{attribute 'GeneratedUsingTerminal: EL5122-0000-0016'}
{attribute addProperty BoxType "EL5122-0000-0016"}
{attribute addProperty Description "EL5122 2Ch. Inc. Encoder 5V (2xAB TTL)"}
{attribute addProperty Physics "KK"}
{attribute addProperty Id "ENC_Status_Channel_1AT %I*ENC_Status_Channel_04F16FC020ENC_Status_Channel_2AT %I*ENC_Status_Channel_04F16FC020ENC_Control_Channel_1AT %Q*ENC_Control_Channel_B930862D10ENC_Control_Channel_2AT %Q*ENC_Control_Channel_B930862D10WcStateAT %I*WcState_9091E0EB2InfoDataAT %I*InfoData_32EB74EA10"}
{attribute addProperty CRC "2132984487"}
{attribute addProperty Size "72"}
TYPE EL5122_7F22C2A7 EXTENDS EtcSlaveTerminalBase_947E5A46 :
STRUCT
	{attribute addProperty Name "ENC_Status_Channel_1"}
	ENC_Status_Channel_1 : ENC_Status_Channel_04F16FC0;
	{attribute addProperty Name "ENC_Status_Channel_2"}
	ENC_Status_Channel_2 : ENC_Status_Channel_04F16FC0;
	{attribute addProperty Name "ENC_Control_Channel_1"}
	ENC_Control_Channel_1 : ENC_Control_Channel_B930862D;
	{attribute addProperty Name "ENC_Control_Channel_2"}
	ENC_Control_Channel_2 : ENC_Control_Channel_B930862D;
	{attribute addProperty Name "WcState"}
	WcState : WcState_9091E0EB;
	{attribute addProperty Name "InfoData"}
	InfoData : InfoData_32EB74EA;
END_STRUCT
END_TYPE

(* stored: Version 1.2.0.0, ProductVersion 3.1.4024.9
   DUT EL5122_7F22C2A7: Id {e13f6fa9-b740-4cf1-8bc8-0b2314c04808} *)
